KUKA KRL data list: ps_a_etb_res_c02.dat

&ACCESS RVO1
&REL 18
&COMMENT Solda Atego ETB
&PARAM DISKPATH = KRC:\R1\Program\OLP
DEFDAT  ps_a_etb_res_c02
;FOLD EXTERNAL DECLARATIONS;%{PE}%MKUKATPBASIS,%CEXT,%VCOMMON,%P
;FOLD GRIPPERTECH EXT
EXT  H50 (INT  :IN,INT  :IN,INT  :IN,GRP_TYP  :IN )
;ENDFOLD (GRIPPERTECH EXT)
;FOLD SPOTTECH EXT
EXT  USERSPOT (S_COMMAND  :IN,SPOT_TYPE  :IN )
;ENDFOLD (SPOTTECH EXT)
;FOLD BASISTECH EXT;%{PE}%MKUKATPBASIS,%CEXT,%VEXT,%P
EXT  BAS (BAS_COMMAND  :IN,REAL  :IN )
DECL INT SUCCESS
;ENDFOLD (BASISTECH EXT)
;FOLD USER EXT;%{E}%MKUKATPUSER,%CEXT,%VEXT,%P
;Make your modifications here

;ENDFOLD (USER EXT)
;ENDFOLD (EXTERNAL DECLARATIONS)


DECL FDAT Fl035={TOOL_NO 3,BASE_NO 3,IPO_FRAME #BASE,POINT2[] " "}
DECL E6POS Xl035={X 584.140991,Y 789.36499,Z 1229.97498,A 158.485001,B 12.9363003,C 166.735794,S 2,T 42}
DECL LDAT LL_OLP8={VEL 2.0,ACC 100.0,APO_DIST 0.0,APO_FAC 0.0,ORI_TYP #VAR,CIRC_TYP #BASE,JERK_FAC 50.0}
DECL FDAT Fl040={TOOL_NO 3,BASE_NO 3,IPO_FRAME #BASE,POINT2[] " "}
DECL E6POS Xl040={X 565.49762,Y 693.462708,Z 1207.63196,A 154.968201,B 9.37270164,C 157.367493,S 18,T 42,E1 0.0,E2 0.0,E3 0.0,E4 0.0,E5 0.0,E6 0.0}
DECL LDAT LL_OLP9={VEL 2.0,ACC 100.0,APO_DIST 0.0,APO_FAC 0.0,ORI_TYP #VAR,CIRC_TYP #BASE,JERK_FAC 50.0}


DECL FDAT Fl045={TOOL_NO 3,BASE_NO 3,IPO_FRAME #BASE,POINT2[] " "}
DECL E6POS Xl045={X 561.989014,Y 691.565002,Z 1096.26794,A 154.969498,B 9.37310028,C 147.3685,S 2,T 42}



DECL LDAT LL_OLP10={VEL 2.0,ACC 100.0,APO_DIST 0.0,APO_FAC 0.0,ORI_TYP #VAR,CIRC_TYP #BASE,JERK_FAC 50.0}
DECL FDAT Fl050={TOOL_NO 3,BASE_NO 3,IPO_FRAME #BASE,POINT2[] " "}
DECL E6POS Xl050={X 563.752014,Y 1566.71301,Z 1132.11096,A 154.969406,B 9.37310028,C 157.3685,S 2,T 42}


DECL LDAT LL_OLP11={VEL 2.0,ACC 100.0,APO_DIST 0.0,APO_FAC 0.0,ORI_TYP #VAR,CIRC_TYP #BASE,JERK_FAC 50.0}
DECL FDAT Fl055={TOOL_NO 3,BASE_NO 3,IPO_FRAME #BASE,POINT2[] " "}
DECL E6POS Xl055={X 878.794006,Y 1301.91504,Z 1209.96802,A -149.936798,B -80.7937012,C 61.0237007,S 2,T 34}
DECL LDAT LL_OLP12={VEL 2.0,ACC 100.0,APO_DIST 0.0,APO_FAC 0.0,ORI_TYP #VAR,CIRC_TYP #BASE,JERK_FAC 50.0}



DECL FDAT Fl060={TOOL_NO 3,BASE_NO 3,IPO_FRAME #BASE,POINT2[] " "}
DECL E6POS Xl060={X 618.291992,Y 968.916992,Z 1209.96594,A -149.936798,B -80.7937012,C 61.0236015,S 2,T 34}
DECL FDAT Fl065={TOOL_NO 3,BASE_NO 3,IPO_FRAME #BASE,POINT2[] " "}
DECL E6POS Xl065={X 584.655212,Y 961.50769,Z 1277.37,A -132.780594,B -83.9849777,C 40.2847786,S 18,T 34,E1 0.0,E2 0.0,E3 0.0,E4 0.0,E5 0.0,E6 0.0}
DECL LDAT LL_OLP14={VEL 2.0,ACC 100.0,APO_DIST 0.0,APO_FAC 0.0,ORI_TYP #VAR,CIRC_TYP #BASE,JERK_FAC 50.0}
DECL FDAT FSWP_60_7788={TOOL_NO 3,BASE_NO 3,IPO_FRAME #BASE,POINT2[] " "}
DECL E6POS XSWP_60_7788={X 594.593811,Y 987.688477,Z 1318.20203,A -158.479996,B -86.9590912,C 65.2634201,S 18,T 34,E1 0.0,E2 0.0,E3 0.0,E4 0.0,E5 0.0,E6 0.0}
DECL LDAT LL_OLP15={VEL 2.0,ACC 100.0,APO_DIST 0.0,APO_FAC 0.0,ORI_TYP #VAR,CIRC_TYP #BASE,JERK_FAC 50.0}
DECL FDAT FSWP_60_7790={TOOL_NO 3,BASE_NO 3,IPO_FRAME #BASE,POINT2[] " ",TQ_STATE FALSE}
DECL E6POS XSWP_60_7790={X 630.833008,Y 988.158813,Z 1320.07104,A 140.789505,B -87.3468933,C 128.901794,S 18,T 34,E1 0.0,E2 0.0,E3 0.0,E4 0.0,E5 0.0,E6 0.0}
DECL LDAT LL_OLP16={VEL 2.0,ACC 100.0,APO_DIST 0.0,APO_FAC 0.0,ORI_TYP #VAR,CIRC_TYP #BASE,JERK_FAC 50.0}
DECL FDAT FSWP_60_7792={TOOL_NO 3,BASE_NO 3,IPO_FRAME #BASE,POINT2[] " "}
DECL E6POS XSWP_60_7792={X 662.220581,Y 987.874329,Z 1321.43994,A 149.062607,B -87.5677567,C 121.765297,S 18,T 34,E1 0.0,E2 0.0,E3 0.0,E4 0.0,E5 0.0,E6 0.0}
DECL LDAT LL_OLP17={VEL 2.0,ACC 100.0,APO_DIST 0.0,APO_FAC 0.0,ORI_TYP #VAR,CIRC_TYP #BASE,JERK_FAC 50.0}
DECL FDAT Fl070={TOOL_NO 3,BASE_NO 3,IPO_FRAME #BASE,POINT2[] " "}
DECL E6POS Xl070={X 658.477173,Y 977.694092,Z 1301.79004,A -86.9980698,B -85.4011383,C -5.58326817,S 18,T 34,E1 0.0,E2 0.0,E3 0.0,E4 0.0,E5 0.0,E6 0.0}
DECL LDAT LL_OLP18={VEL 2.0,ACC 100.0,APO_DIST 0.0,APO_FAC 0.0,ORI_TYP #VAR,CIRC_TYP #BASE,JERK_FAC 50.0}

DECL FDAT Fl075={TOOL_NO 3,BASE_NO 3,IPO_FRAME #BASE,POINT2[] " "}



DECL E6POS Xl075={X 670.585022,Y 967.37323,Z 1219.30298,A -89.5080719,B -85.5535965,C 0.906028271,S 18,T 34,E1 0.0,E2 0.0,E3 0.0,E4 0.0,E5 0.0,E6 0.0}
DECL LDAT LL_OLP19={VEL 2.0,ACC 100.0,APO_DIST 10.0,APO_FAC 0.0,ORI_TYP #VAR,CIRC_TYP #BASE,JERK_FAC 50.0}






DECL FDAT Fl080={TOOL_NO 3,BASE_NO 3,IPO_FRAME #BASE,POINT2[] " "}
DECL E6POS Xl080={X 704.95752,Y 967.856384,Z 1264.87,A -14.49963,B -74.4627228,C -73.6447296,S 18,T 34,E1 0.0,E2 0.0,E3 0.0,E4 0.0,E5 0.0,E6 0.0}
DECL LDAT LL_OLP20={VEL 2.0,ACC 100.0,APO_DIST 10.0,APO_FAC 0.0,ORI_TYP #VAR,CIRC_TYP #BASE,JERK_FAC 50.0}
DECL FDAT Fl085={TOOL_NO 3,BASE_NO 3,IPO_FRAME #BASE,POINT2[] " "}
DECL E6POS Xl085={X 715.177124,Y 970.295776,Z 1286.88904,A -14.4969301,B -74.4632263,C -73.6462326,S 18,T 34,E1 0.0,E2 0.0,E3 0.0,E4 0.0,E5 0.0,E6 0.0}
DECL LDAT LL_OLP21={VEL 2.0,ACC 100.0,APO_DIST 0.0,APO_FAC 0.0,ORI_TYP #VAR,CIRC_TYP #BASE,JERK_FAC 50.0}
DECL FDAT FSWP_60_7796={TOOL_NO 3,BASE_NO 3,IPO_FRAME #BASE,POINT2[] " "}
DECL E6POS XSWP_60_7796={X 735.90741,Y 986.652527,Z 1321.86902,A 8.92792034,B -75.0170135,C -96.2646103,S 18,T 34,E1 0.0,E2 0.0,E3 0.0,E4 0.0,E5 0.0,E6 0.0}
DECL LDAT LL_OLP22={VEL 2.0,ACC 100.0,APO_DIST 0.0,APO_FAC 0.0,ORI_TYP #VAR,CIRC_TYP #BASE,JERK_FAC 50.0}
DECL FDAT FSWP_60_7798={TOOL_NO 3,BASE_NO 3,IPO_FRAME #BASE,POINT2[] " "}
DECL E6POS XSWP_60_7798={X 779.640076,Y 986.603088,Z 1321.69299,A 4.67745781,B -75.0973206,C -92.1623993,S 18,T 34,E1 0.0,E2 0.0,E3 0.0,E4 0.0,E5 0.0,E6 0.0}
DECL LDAT LL_OLP23={VEL 2.0,ACC 100.0,APO_DIST 0.0,APO_FAC 0.0,ORI_TYP #VAR,CIRC_TYP #BASE,JERK_FAC 50.0}
DECL FDAT FSWP_60_7800={TOOL_NO 3,BASE_NO 3,IPO_FRAME #BASE,POINT2[] " "}
DECL E6POS XSWP_60_7800={X 825.9328,Y 985.137573,Z 1320.76904,A 4.2847209,B -75.2969131,C -91.1992035,S 18,T 34,E1 0.0,E2 0.0,E3 0.0,E4 0.0,E5 0.0,E6 0.0}
DECL LDAT LL_OLP24={VEL 2.0,ACC 100.0,APO_DIST 0.0,APO_FAC 0.0,ORI_TYP #VAR,CIRC_TYP #BASE,JERK_FAC 50.0}
DECL FDAT FSWP_60_7802={TOOL_NO 3,BASE_NO 3,IPO_FRAME #BASE,POINT2[] " "}
DECL E6POS XSWP_60_7802={X 869.143188,Y 986.01178,Z 1322.323,A -7.07776499,B -75.2145462,C -79.7799606,S 18,T 34,E1 0.0,E2 0.0,E3 0.0,E4 0.0,E5 0.0,E6 0.0}
DECL LDAT LL_OLP25={VEL 2.0,ACC 100.0,APO_DIST 0.0,APO_FAC 0.0,ORI_TYP #VAR,CIRC_TYP #BASE,JERK_FAC 50.0}
DECL FDAT FSWP_60_7804={TOOL_NO 3,BASE_NO 3,IPO_FRAME #BASE,POINT2[] " "}
DECL E6POS XSWP_60_7804={X 921.059021,Y 987.353088,Z 1322.45996,A -5.14408016,B -75.1806793,C -81.9926834,S 18,T 34,E1 0.0,E2 0.0,E3 0.0,E4 0.0,E5 0.0,E6 0.0}
DECL LDAT LL_OLP26={VEL 2.0,ACC 100.0,APO_DIST 0.0,APO_FAC 0.0,ORI_TYP #VAR,CIRC_TYP #BASE,JERK_FAC 50.0}
DECL FDAT FSWP_60_7808={TOOL_NO 3,BASE_NO 3,IPO_FRAME #BASE,POINT2[] " "}
DECL E6POS XSWP_60_7808={X 1013.84802,Y 985.960999,Z 1321.65198,A -9.0603056,B -74.9901505,C -78.2635727,S 18,T 34,E1 0.0,E2 0.0,E3 0.0,E4 0.0,E5 0.0,E6 0.0}
DECL LDAT LL_OLP27={VEL 2.0,ACC 100.0,APO_DIST 0.0,APO_FAC 0.0,ORI_TYP #VAR,CIRC_TYP #BASE,JERK_FAC 50.0}
DECL FDAT FSWP_60_7810={TOOL_NO 3,BASE_NO 3,IPO_FRAME #BASE,POINT2[] " "}
DECL E6POS XSWP_60_7810={X 1060.09204,Y 986.898987,Z 1321.53003,A -9.69570732,B -74.9384232,C -77.7038574,S 18,T 34,E1 0.0,E2 0.0,E3 0.0,E4 0.0,E5 0.0,E6 0.0}
DECL LDAT LL_OLP28={VEL 2.0,ACC 100.0,APO_DIST 0.0,APO_FAC 0.0,ORI_TYP #VAR,CIRC_TYP #BASE,JERK_FAC 50.0}
DECL FDAT FSWP_60_7812={TOOL_NO 3,BASE_NO 3,IPO_FRAME #BASE,POINT2[] " "}
DECL E6POS XSWP_60_7812={X 1103.44104,Y 986.481995,Z 1321.01294,A -11.51863,B -74.7812805,C -76.1086578,S 18,T 34,E1 0.0,E2 0.0,E3 0.0,E4 0.0,E5 0.0,E6 0.0}
DECL LDAT LL_OLP29={VEL 2.0,ACC 100.0,APO_DIST 0.0,APO_FAC 0.0,ORI_TYP #VAR,CIRC_TYP #BASE,JERK_FAC 50.0}
DECL FDAT FSWP_60_7814={TOOL_NO 3,BASE_NO 3,IPO_FRAME #BASE,POINT2[] " "}
DECL E6POS XSWP_60_7814={X 1146.948,Y 986.203918,Z 1319.48206,A -9.90011024,B -74.91008,C -77.5603333,S 18,T 34,E1 0.0,E2 0.0,E3 0.0,E4 0.0,E5 0.0,E6 0.0}
DECL LDAT LL_OLP30={VEL 2.0,ACC 100.0,APO_DIST 0.0,APO_FAC 0.0,ORI_TYP #VAR,CIRC_TYP #BASE,JERK_FAC 50.0}
DECL FDAT FSWP_60_7816={TOOL_NO 3,BASE_NO 3,IPO_FRAME #BASE,POINT2[] " "}
DECL E6POS XSWP_60_7816={X 1193.84399,Y 985.979675,Z 1318.43506,A -3.22997093,B -75.0365219,C -84.5187073,S 18,T 34,E1 0.0,E2 0.0,E3 0.0,E4 0.0,E5 0.0,E6 0.0}
DECL LDAT LL_OLP31={VEL 2.0,ACC 100.0,APO_DIST 0.0,APO_FAC 0.0,ORI_TYP #VAR,CIRC_TYP #BASE,JERK_FAC 50.0}
DECL FDAT Fl090={TOOL_NO 3,BASE_NO 3,IPO_FRAME #BASE,POINT2[] " "}
DECL E6POS Xl090={X 1197.92505,Y 977.659119,Z 1291.51294,A -14.5019197,B -74.4627228,C -73.6420135,S 18,T 34,E1 0.0,E2 0.0,E3 0.0,E4 0.0,E5 0.0,E6 0.0}
DECL LDAT LL_OLP32={VEL 2.0,ACC 100.0,APO_DIST 0.0,APO_FAC 0.0,ORI_TYP #VAR,CIRC_TYP #BASE,JERK_FAC 50.0}
DECL FDAT Fl095={TOOL_NO 3,BASE_NO 3,IPO_FRAME #BASE,POINT2[] " "}
DECL E6POS Xl095={X 1176.53894,Y 994.848877,Z 1208.64905,A -44.5544205,B -83.8928528,C -43.9489098,S 18,T 34,E1 0.0,E2 0.0,E3 0.0,E4 0.0,E5 0.0,E6 0.0}
DECL LDAT LL_OLP33={VEL 2.0,ACC 100.0,APO_DIST 0.0,APO_FAC 0.0,ORI_TYP #VAR,CIRC_TYP #BASE,JERK_FAC 50.0}















DECL FDAT Fl100={TOOL_NO 3,BASE_NO 3,IPO_FRAME #BASE,POINT2[] " "}
DECL E6POS Xl100={X 795.249023,Y 1246.63,Z 1059.69897,A -149.936401,B -80.7937012,C 61.023201,S 2,T 34}
DECL LDAT LL_OLP34={VEL 2.0,ACC 100.0,APO_DIST 10.0,APO_FAC 0.0,ORI_TYP #VAR,CIRC_TYP #BASE,JERK_FAC 50.0}
DECL FDAT Fl105={TOOL_NO 3,BASE_NO 3,IPO_FRAME #BASE,POINT2[] " "}
DECL E6POS Xl105={X 1304.354,Y 1333.35901,Z 23.5259991,A 180.0,B -37.3134003,C 90.0,S 2,T 34}
DECL LDAT LL_OLP35={VEL 2.0,ACC 100.0,APO_DIST 30.0,APO_FAC 0.0,ORI_TYP #VAR,CIRC_TYP #BASE,JERK_FAC 50.0}

DECL FDAT Fl120={TOOL_NO 3,BASE_NO 3,IPO_FRAME #BASE,POINT2[] " "}

DECL E6POS Xl120={X 1303.89905,Y 1020.01202,Z 107.1138,A 179.976105,B -22.3131905,C 89.996582,S 18,T 34,E1 0.0,E2 0.0,E3 0.0,E4 0.0,E5 0.0,E6 0.0}
DECL LDAT LL_OLP38={VEL 2.0,ACC 100.0,APO_DIST 0.0,APO_FAC 0.0,ORI_TYP #VAR,CIRC_TYP #BASE,JERK_FAC 50.0}

DECL FDAT FSWP_60_7488={TOOL_NO 3,BASE_NO 3,IPO_FRAME #BASE,POINT2[] " "}

DECL E6POS XSWP_60_7488={X 1311.29602,Y 1033.21301,Z 114.044098,A 179.174393,B -22.3031502,C 90.7230225,S 18,T 34,E1 0.0,E2 0.0,E3 0.0,E4 0.0,E5 0.0,E6 0.0}
DECL LDAT LL_OLP39={VEL 2.0,ACC 100.0,APO_DIST 0.0,APO_FAC 0.0,ORI_TYP #VAR,CIRC_TYP #BASE,JERK_FAC 50.0}

DECL FDAT FSWP_60_7490={TOOL_NO 3,BASE_NO 3,IPO_FRAME #BASE,POINT2[] " "}

DECL E6POS XSWP_60_7490={X 1343.07202,Y 1031.32202,Z 114.458504,A 179.979507,B -22.3129196,C 90.9136505,S 18,T 34,E1 0.0,E2 0.0,E3 0.0,E4 0.0,E5 0.0,E6 0.0}
DECL LDAT LL_OLP40={VEL 2.0,ACC 100.0,APO_DIST 0.0,APO_FAC 0.0,ORI_TYP #VAR,CIRC_TYP #BASE,JERK_FAC 50.0}

DECL FDAT FSWP_60_7492={TOOL_NO 3,BASE_NO 3,IPO_FRAME #BASE,POINT2[] " "}

DECL E6POS XSWP_60_7492={X 1374.18799,Y 1032.23499,Z 114.821899,A -179.808701,B -22.2939205,C 89.9696426,S 18,T 34,E1 0.0,E2 0.0,E3 0.0,E4 0.0,E5 0.0,E6 0.0}
DECL LDAT LL_OLP41={VEL 2.0,ACC 100.0,APO_DIST 0.0,APO_FAC 0.0,ORI_TYP #VAR,CIRC_TYP #BASE,JERK_FAC 50.0}

DECL FDAT Fl125={TOOL_NO 3,BASE_NO 3,IPO_FRAME #BASE,POINT2[] " "}


DECL E6POS Xl125={X 1397.44604,Y 1024.76294,Z 95.6467438,A 179.9758,B -17.5534992,C 89.9962769,S 18,T 34,E1 0.0,E2 0.0,E3 0.0,E4 0.0,E5 0.0,E6 0.0}
DECL LDAT LL_OLP42={VEL 2.0,ACC 100.0,APO_DIST 0.0,APO_FAC 0.0,ORI_TYP #VAR,CIRC_TYP #BASE,JERK_FAC 50.0}
DECL FDAT Fl130={TOOL_NO 3,BASE_NO 3,IPO_FRAME #BASE,POINT2[] " "}
DECL E6POS Xl130={X 1469.67896,Y 1023.99103,Z 98.598999,A 179.975601,B -17.0133991,C 89.9968033,S 2,T 34}
DECL LDAT LL_OLP43={VEL 2.0,ACC 100.0,APO_DIST 0.0,APO_FAC 0.0,ORI_TYP #VAR,CIRC_TYP #BASE,JERK_FAC 50.0}



DECL FDAT FSWP_60_7496={TOOL_NO 3,BASE_NO 3,IPO_FRAME #BASE,POINT2[] " "}

DECL E6POS XSWP_60_7496={X 1451.85803,Y 1028.74304,Z 116.249001,A 179.984207,B -21.8110695,C 94.6477966,S 18,T 42,E1 0.0,E2 0.0,E3 0.0,E4 0.0,E5 0.0,E6 0.0}
DECL LDAT LL_OLP44={VEL 2.0,ACC 100.0,APO_DIST 0.0,APO_FAC 0.0,ORI_TYP #VAR,CIRC_TYP #BASE,JERK_FAC 50.0}

DECL FDAT FSWP_60_7498={TOOL_NO 3,BASE_NO 3,IPO_FRAME #BASE,POINT2[] " "}


DECL E6POS XSWP_60_7498={X 1491.27698,Y 1028.06201,Z 116.260399,A 179.982605,B -21.8108807,C 94.0462494,S 18,T 42,E1 0.0,E2 0.0,E3 0.0,E4 0.0,E5 0.0,E6 0.0}
DECL LDAT LL_OLP45={VEL 2.0,ACC 100.0,APO_DIST 0.0,APO_FAC 0.0,ORI_TYP #VAR,CIRC_TYP #BASE,JERK_FAC 50.0}
DECL FDAT FSWP_60_7500={TOOL_NO 3,BASE_NO 3,IPO_FRAME #BASE,POINT2[] " "}
DECL E6POS XSWP_60_7500={X 1538.92004,Y 1026.06396,Z 113.879898,A -179.763596,B -29.0331993,C 93.614418,S 18,T 34,E1 0.0,E2 0.0,E3 0.0,E4 0.0,E5 0.0,E6 0.0}
DECL LDAT LL_OLP46={VEL 2.0,ACC 100.0,APO_DIST 0.0,APO_FAC 0.0,ORI_TYP #VAR,CIRC_TYP #BASE,JERK_FAC 50.0}

DECL FDAT Fl140={TOOL_NO 3,BASE_NO 3,IPO_FRAME #BASE,POINT2[] " "}
DECL PDAT PP_OLP2={VEL 100.0,ACC 100.0,APO_DIST 0.0,APO_MODE #CDIS}
DECL E6POS Xl140={X 1610.60205,Y 1139.57495,Z 45.987999,A 179.975998,B -22.3132992,C 89.9968033,S 2,T 34}
DECL BASIS_SUGG_T LAST_BASIS={POINT1[] "PS01010001              ",POINT2[] "PS01010001              ",CP_PARAMS[] "CPDAT0                  ",PTP_PARAMS[] "PDAT0                   ",CONT[] "                        ",CP_VEL[] "2                       ",PTP_VEL[] " 100                    ",SPL_NAME[] "S0                      "}
DECL PDAT PP_OLP4={VEL 100.0,ACC 100.0,APO_DIST 30.0,APO_MODE #CDIS}
DECL E6POS Xl006={X 1083.797,Y 1451.30701,Z 836.236023,A 174.173294,B -30.1965008,C 118.184799,S 2,T 42}
DECL FDAT Fl006={TOOL_NO 3,BASE_NO 3,IPO_FRAME #BASE,POINT2[] " "}
DECL E6POS Xl011={X 563.747314,Y 1566.72302,Z 1132.10205,A 154.969299,B 9.37345028,C 157.368103,S 18,T 42,E1 0.0,E2 0.0,E3 0.0,E4 0.0,E5 0.0,E6 0.0}
DECL FDAT Fl011={TOOL_NO 3,BASE_NO 3,IPO_FRAME #BASE,POINT2[] " ",TQ_STATE FALSE}
DECL LDAT LL_OLP49={VEL 2.0,ACC 100.0,APO_DIST 0.0,APO_FAC 0.0,ORI_TYP #VAR,CIRC_TYP #BASE,JERK_FAC 50.0}
DECL E6POS Xl016={X 561.989014,Y 691.565002,Z 1096.26794,A 154.969498,B 9.37310028,C 147.3685,S 2,T 42}
DECL FDAT Fl016={TOOL_NO 3,BASE_NO 3,IPO_FRAME #BASE,POINT2[] " "}
DECL PDAT PP_OLP5={VEL 100.0,ACC 100.0,APO_DIST 0.0}
DECL E6POS Xl021={X 563.750977,Y 693.715027,Z 1132.11096,A 154.969406,B 9.37310028,C 157.3685,S 2,T 42}
DECL FDAT Fl021={TOOL_NO 3,BASE_NO 3,IPO_FRAME #BASE,POINT2[] " "}
DECL LDAT LL_OLP50={VEL 2.0,ACC 100.0,APO_DIST 30.0,APO_FAC 0.0,ORI_TYP #VAR,CIRC_TYP #BASE,JERK_FAC 50.0}
DECL E6POS Xl026={X 584.140991,Y 789.36499,Z 1229.97498,A 158.485001,B 12.9363003,C 166.735794,S 2,T 42}
DECL FDAT Fl026={TOOL_NO 3,BASE_NO 3,IPO_FRAME #BASE,POINT2[] " "}












DECL LDAT LL_OLP51={VEL 2.0,ACC 100.0,APO_DIST 0.0,APO_FAC 0.0,ORI_TYP #VAR,CIRC_TYP #BASE,JERK_FAC 50.0}
DECL E6POS Xl031={X 349.9328,Y 278.265503,Z 1120.06702,A 150.3909,B 43.1627502,C 155.956406,S 18,T 42,E1 0.0,E2 0.0,E3 0.0,E4 0.0,E5 0.0,E6 0.0}
DECL FDAT Fl031={TOOL_NO 3,BASE_NO 3,IPO_FRAME #BASE,POINT2[] " "}
DECL PDAT PP_OLP6={VEL 100.0,ACC 100.0,APO_DIST 0.0}
DECL E6POS Xl036={X 305.381195,Y 288.633514,Z 1051.12598,A 147.643494,B 47.8914604,C 153.831299,S 18,T 42,E1 0.0,E2 0.0,E3 0.0,E4 0.0,E5 0.0,E6 0.0}
DECL FDAT Fl036={TOOL_NO 3,BASE_NO 3,IPO_FRAME #BASE,POINT2[] " "}
DECL PDAT PP_OLP7={VEL 100.0,ACC 100.0,APO_DIST 10.0,APO_MODE #CDIS}
DECL E6POS Xl041={X 103.434502,Y 364.44751,Z 683.522705,A 164.801605,B 79.9912796,C 167.123993,S 18,T 42,E1 0.0,E2 0.0,E3 0.0,E4 0.0,E5 0.0,E6 0.0}
DECL FDAT Fl041={TOOL_NO 3,BASE_NO 3,IPO_FRAME #BASE,POINT2[] " "}
DECL LDAT LL_OLP52={VEL 2.0,ACC 100.0,APO_DIST 0.0,APO_FAC 0.0,ORI_TYP #VAR,CIRC_TYP #BASE,JERK_FAC 50.0}
DECL E6POS Xl046={X 91.8286896,Y 379.290894,Z 653.815796,A 159.358994,B 82.8835907,C 161.735306,S 18,T 42,E1 0.0,E2 0.0,E3 0.0,E4 0.0,E5 0.0,E6 0.0}
DECL FDAT Fl046={TOOL_NO 3,BASE_NO 3,IPO_FRAME #BASE,POINT2[] " "}
DECL LDAT LL_OLP53={VEL 2.0,ACC 100.0,APO_DIST 0.0,APO_FAC 0.0,ORI_TYP #VAR,CIRC_TYP #BASE,JERK_FAC 50.0}
DECL E6POS XSWP_60_7880={X 93.7982178,Y 380.760986,Z 613.06543,A 159.360794,B 82.8838272,C 161.736404,S 18,T 42,E1 0.0,E2 0.0,E3 0.0,E4 0.0,E5 0.0,E6 0.0}
DECL FDAT FSWP_60_7880={TOOL_NO 3,BASE_NO 3,IPO_FRAME #BASE,POINT2[] " "}
DECL LDAT LL_OLP54={VEL 2.0,ACC 100.0,APO_DIST 0.0,APO_FAC 0.0,ORI_TYP #VAR,CIRC_TYP #BASE,JERK_FAC 50.0}
DECL E6POS XSWP_60_7882={X 95.1983414,Y 412.033203,Z 612.224121,A 159.370499,B 82.8822937,C 161.745895,S 18,T 42,E1 0.0,E2 0.0,E3 0.0,E4 0.0,E5 0.0,E6 0.0}
DECL FDAT FSWP_60_7882={TOOL_NO 3,BASE_NO 3,IPO_FRAME #BASE,POINT2[] " "}
DECL LDAT LL_OLP55={VEL 2.0,ACC 100.0,APO_DIST 0.0,APO_FAC 0.0,ORI_TYP #VAR,CIRC_TYP #BASE,JERK_FAC 50.0}
DECL E6POS XSWP_60_7886={X 98.8377228,Y 478.136993,Z 615.090515,A 158.5354,B 82.6687012,C 159.334305,S 18,T 42,E1 0.0,E2 0.0,E3 0.0,E4 0.0,E5 0.0,E6 0.0}
DECL FDAT FSWP_60_7886={TOOL_NO 3,BASE_NO 3,IPO_FRAME #BASE,POINT2[] " "}
DECL LDAT LL_OLP56={VEL 2.0,ACC 100.0,APO_DIST 0.0,APO_FAC 0.0,ORI_TYP #VAR,CIRC_TYP #BASE,JERK_FAC 50.0}
DECL E6POS XSWP_60_7888={X 100.442497,Y 513.4646,Z 616.12793,A 159.082596,B 82.9018936,C 159.794601,S 18,T 42,E1 0.0,E2 0.0,E3 0.0,E4 0.0,E5 0.0,E6 0.0}
DECL FDAT FSWP_60_7888={TOOL_NO 3,BASE_NO 3,IPO_FRAME #BASE,POINT2[] " "}
DECL LDAT LL_OLP57={VEL 2.0,ACC 100.0,APO_DIST 0.0,APO_FAC 0.0,ORI_TYP #VAR,CIRC_TYP #BASE,JERK_FAC 50.0}
DECL E6POS XSWP_60_7990={X 102.522003,Y 545.988403,Z 614.039917,A 160.234299,B 82.879837,C 161.132095,S 18,T 42,E1 0.0,E2 0.0,E3 0.0,E4 0.0,E5 0.0,E6 0.0}
DECL FDAT FSWP_60_7990={TOOL_NO 3,BASE_NO 3,IPO_FRAME #BASE,POINT2[] " "}
DECL LDAT LL_OLP58={VEL 2.0,ACC 100.0,APO_DIST 0.0,APO_FAC 0.0,ORI_TYP #VAR,CIRC_TYP #BASE,JERK_FAC 50.0}
DECL E6POS XSWP_60_7892={X 103.919098,Y 574.488892,Z 615.100891,A 159.7061,B 82.8799286,C 161.684998,S 18,T 42,E1 0.0,E2 0.0,E3 0.0,E4 0.0,E5 0.0,E6 0.0}
DECL FDAT FSWP_60_7892={TOOL_NO 3,BASE_NO 3,IPO_FRAME #BASE,POINT2[] " "}
DECL LDAT LL_OLP59={VEL 2.0,ACC 100.0,APO_DIST 0.0,APO_FAC 0.0,ORI_TYP #VAR,CIRC_TYP #BASE,JERK_FAC 50.0}
DECL E6POS XSWP_60_7896={X 108.416,Y 646.456177,Z 614.435181,A 159.410507,B 82.8830185,C 161.785904,S 18,T 42,E1 0.0,E2 0.0,E3 0.0,E4 0.0,E5 0.0,E6 0.0}
DECL FDAT FSWP_60_7896={TOOL_NO 3,BASE_NO 3,IPO_FRAME #BASE,POINT2[] " "}
DECL LDAT LL_OLP60={VEL 2.0,ACC 100.0,APO_DIST 0.0,APO_FAC 0.0,ORI_TYP #VAR,CIRC_TYP #BASE,JERK_FAC 50.0}
DECL E6POS XSWP_60_7898={X 111.716202,Y 682.766418,Z 615.322815,A 159.398407,B 82.8831482,C 161.775604,S 18,T 42,E1 0.0,E2 0.0,E3 0.0,E4 0.0,E5 0.0,E6 0.0}
DECL FDAT FSWP_60_7898={TOOL_NO 3,BASE_NO 3,IPO_FRAME #BASE,POINT2[] " "}
DECL LDAT LL_OLP61={VEL 2.0,ACC 100.0,APO_DIST 0.0,APO_FAC 0.0,ORI_TYP #VAR,CIRC_TYP #BASE,JERK_FAC 50.0}
DECL E6POS XSWP_60_7900={X 114.766197,Y 718.722412,Z 616.54657,A 159.434402,B 82.8802872,C 161.813995,S 18,T 42,E1 0.0,E2 0.0,E3 0.0,E4 0.0,E5 0.0,E6 0.0}
DECL FDAT FSWP_60_7900={TOOL_NO 3,BASE_NO 3,IPO_FRAME #BASE,POINT2[] " "}
DECL LDAT LL_OLP62={VEL 2.0,ACC 100.0,APO_DIST 0.0,APO_FAC 0.0,ORI_TYP #VAR,CIRC_TYP #BASE,JERK_FAC 50.0}
DECL E6POS XSWP_60_7902={X 119.6847,Y 754.768677,Z 617.763794,A 159.414795,B 82.8860092,C 161.790604,S 18,T 42,E1 0.0,E2 0.0,E3 0.0,E4 0.0,E5 0.0,E6 0.0}
DECL FDAT FSWP_60_7902={TOOL_NO 3,BASE_NO 3,IPO_FRAME #BASE,POINT2[] " "}
DECL LDAT LL_OLP63={VEL 2.0,ACC 100.0,APO_DIST 0.0,APO_FAC 0.0,ORI_TYP #VAR,CIRC_TYP #BASE,JERK_FAC 50.0}
DECL E6POS XSWP_60_7904={X 124.1399,Y 792.107971,Z 618.820129,A 159.417999,B 82.8863525,C 161.793106,S 18,T 42,E1 0.0,E2 0.0,E3 0.0,E4 0.0,E5 0.0,E6 0.0}
DECL FDAT FSWP_60_7904={TOOL_NO 3,BASE_NO 3,IPO_FRAME #BASE,POINT2[] " "}
DECL LDAT LL_OLP64={VEL 2.0,ACC 100.0,APO_DIST 0.0,APO_FAC 0.0,ORI_TYP #VAR,CIRC_TYP #BASE,JERK_FAC 50.0}
DECL E6POS XSWP_60_7906={X 132.870697,Y 841.648804,Z 621.361816,A 159.395203,B 82.8851624,C 161.773804,S 18,T 42,E1 0.0,E2 0.0,E3 0.0,E4 0.0,E5 0.0,E6 0.0}
DECL FDAT FSWP_60_7906={TOOL_NO 3,BASE_NO 3,IPO_FRAME #BASE,POINT2[] " "}
DECL LDAT LL_OLP65={VEL 2.0,ACC 100.0,APO_DIST 0.0,APO_FAC 0.0,ORI_TYP #VAR,CIRC_TYP #BASE,JERK_FAC 50.0}
DECL E6POS XSWP_60_7908={X 139.911102,Y 879.169617,Z 618.96582,A 159.404099,B 82.897049,C 167.300797,S 18,T 42,E1 0.0,E2 0.0,E3 0.0,E4 0.0,E5 0.0,E6 0.0}
DECL FDAT FSWP_60_7908={TOOL_NO 3,BASE_NO 3,IPO_FRAME #BASE,POINT2[] " "}
DECL E6POS Xl051={X 137.945007,Y 854.049988,Z 676.479004,A 164.794098,B 79.9898987,C 167.113907,S 2,T 42}
DECL FDAT Fl051={TOOL_NO 3,BASE_NO 3,IPO_FRAME #BASE,POINT2[] " "}
DECL SPOT_TYPE SNORMAL={GUN 1,PAIR #FIRST,RETR #OPN,CLO_TM 0,PGNO1 1,PRESS1 0.0,PGNO2 0,PRESS2 0.0}
DECL E6POS XP3={X 567.326416,Y 409.623993,Z 1234.31702,A 158.465195,B 12.93505,C 166.748199,S 18,T 42,E1 0.0,E2 0.0,E3 0.0,E4 0.0,E5 0.0,E6 0.0}
DECL FDAT FP3={TOOL_NO 3,BASE_NO 3,IPO_FRAME #BASE,POINT2[] " ",TQ_STATE FALSE}
DECL LDAT LCPDAT2={VEL 2.0,ACC 100.0,APO_DIST 10.0,APO_FAC 50.0,AXIS_VEL 100.0,AXIS_ACC 100.0,ORI_TYP #VAR,CIRC_TYP #BASE,JERK_FAC 50.0,GEAR_JERK 50.0,EXAX_IGN 0}
DECL E6POS XP6={X 558.674316,Y 257.743713,Z 1366.94299,A 155.132797,B 22.3248005,C 163.028503,S 18,T 42,E1 0.0,E2 0.0,E3 0.0,E4 0.0,E5 0.0,E6 0.0}
DECL FDAT FP6={TOOL_NO 3,BASE_NO 3,IPO_FRAME #BASE,POINT2[] " ",TQ_STATE FALSE}
DECL LDAT LCPDAT5={VEL 2.0,ACC 100.0,APO_DIST 100.0,APO_FAC 50.0,AXIS_VEL 100.0,AXIS_ACC 100.0,ORI_TYP #VAR,CIRC_TYP #BASE,JERK_FAC 50.0,GEAR_JERK 50.0,EXAX_IGN 0}
DECL E6POS XP7={X 622.916321,Y 355.254211,Z 1422.57605,A 157.948105,B 12.9317598,C 166.758606,S 18,T 42,E1 0.0,E2 0.0,E3 0.0,E4 0.0,E5 0.0,E6 0.0}
DECL FDAT FP7={TOOL_NO 3,BASE_NO 3,IPO_FRAME #BASE,POINT2[] " ",TQ_STATE FALSE}
DECL LDAT LCPDAT6={VEL 2.0,ACC 100.0,APO_DIST 100.0,APO_FAC 50.0,AXIS_VEL 100.0,AXIS_ACC 100.0,ORI_TYP #VAR,CIRC_TYP #BASE,JERK_FAC 50.0,GEAR_JERK 50.0,EXAX_IGN 0}
DECL E6POS XP8={X 407.655396,Y 277.337799,Z 1190.83606,A 150.367401,B 35.5736084,C 156.603897,S 18,T 42,E1 0.0,E2 0.0,E3 0.0,E4 0.0,E5 0.0,E6 0.0}
DECL FDAT FP8={TOOL_NO 3,BASE_NO 3,IPO_FRAME #BASE,POINT2[] " ",TQ_STATE FALSE}
DECL LDAT LCPDAT7={VEL 2.0,ACC 100.0,APO_DIST 100.0,APO_FAC 50.0,AXIS_VEL 100.0,AXIS_ACC 100.0,ORI_TYP #VAR,CIRC_TYP #BASE,JERK_FAC 50.0,GEAR_JERK 50.0,EXAX_IGN 0}


DECL E6POS XP11={X 1560.58704,Y 1009.72302,Z 65.5483475,A 179.964401,B -43.8393517,C 90.9567795,S 18,T 34,E1 0.0,E2 0.0,E3 0.0,E4 0.0,E5 0.0,E6 0.0}
DECL FDAT FP11={TOOL_NO 3,BASE_NO 3,IPO_FRAME #BASE,POINT2[] " ",TQ_STATE FALSE}

DECL LDAT LCPDAT10={VEL 2.0,ACC 100.0,APO_DIST 100.0,APO_FAC 50.0,AXIS_VEL 100.0,AXIS_ACC 100.0,ORI_TYP #VAR,CIRC_TYP #BASE,JERK_FAC 50.0,GEAR_JERK 50.0,EXAX_IGN 0}
DECL SPOT_SUGG_T LAST_SPOT={GUN[] "1                       ",RETR_CMD[] "#OPN                    ",CHOISE[] "#FIRST                  ",CLO_TM[] "0                       ",PGNO1[] "1                       ",PRESS1[] "0                       ",PGNO2[] "1                       ",PRESS2[] "0                       ",SPOT_PARAMS[] "NORMAL                  "}
DECL E6POS XP14={X 1610.68799,Y 1340.54297,Z 45.7100296,A 179.967102,B -22.3057804,C 90.001152,S 18,T 34,E1 0.0,E2 0.0,E3 0.0,E4 0.0,E5 0.0,E6 0.0}
DECL FDAT FP14={TOOL_NO 3,BASE_NO 3,IPO_FRAME #BASE,POINT2[] " ",TQ_STATE FALSE}
DECL PDAT PPDAT5={VEL 100.0,ACC 95.0,APO_DIST 100.0,APO_MODE #CDIS,GEAR_JERK 50.0}
DECL E6POS XP16={X 1711.52502,Y 2023.51099,Z 556.947876,A -175.166397,B -41.1158485,C 86.8608398,S 18,T 34,E1 0.0,E2 0.0,E3 0.0,E4 0.0,E5 0.0,E6 0.0}
DECL FDAT FP16={TOOL_NO 3,BASE_NO 3,IPO_FRAME #BASE,POINT2[] " ",TQ_STATE FALSE}
DECL PDAT PPDAT7={VEL 100.0,ACC 100.0,APO_DIST 100.0,APO_MODE #CDIS,GEAR_JERK 50.0}
DECL E6POS XP17={X 1711.651,Y 2023.50098,Z 556.917297,A -175.160202,B -41.1122093,C 86.8591003,S 18,T 42,E1 0.0,E2 0.0,E3 0.0,E4 0.0,E5 0.0,E6 0.0}


DECL FDAT FP17={TOOL_NO 3,BASE_NO 3,IPO_FRAME #BASE,POINT2[] " ",TQ_STATE FALSE}
DECL PDAT PPDAT8={VEL 100.0,ACC 100.0,APO_DIST 100.0,APO_MODE #CDIS,GEAR_JERK 50.0}
DECL LDAT LCPDAT11={VEL 2.0,ACC 100.0,APO_DIST 10.0,APO_FAC 50.0,AXIS_VEL 100.0,AXIS_ACC 100.0,ORI_TYP #VAR,CIRC_TYP #BASE,JERK_FAC 50.0,GEAR_JERK 50.0,EXAX_IGN 0}
DECL E6POS XP18={X 60.9463196,Y 487.706207,Z 619.175598,A 160.159195,B 82.8793716,C 161.610504,S 18,T 42,E1 0.0,E2 0.0,E3 0.0,E4 0.0,E5 0.0,E6 0.0}
DECL FDAT FP18={TOOL_NO 3,BASE_NO 3,IPO_FRAME #BASE,POINT2[] " ",TQ_STATE FALSE}
DECL LDAT LCPDAT12={VEL 2.0,ACC 100.0,APO_DIST 10.0,APO_FAC 50.0,AXIS_VEL 100.0,AXIS_ACC 100.0,ORI_TYP #VAR,CIRC_TYP #BASE,JERK_FAC 50.0,GEAR_JERK 50.0,EXAX_IGN 0}

DECL E6POS XP19={X 128.315308,Y 824.686523,Z 636.831726,A 156.575699,B 83.7855835,C 158.972504,S 18,T 42,E1 0.0,E2 0.0,E3 0.0,E4 0.0,E5 0.0,E6 0.0}

DECL FDAT FP19={TOOL_NO 3,BASE_NO 3,IPO_FRAME #BASE,POINT2[] " ",TQ_STATE FALSE}

DECL LDAT LL_OLP68={VEL 2.0,ACC 100.0,APO_DIST 10.0,APO_FAC 0.0,ORI_TYP #VAR,CIRC_TYP #BASE,JERK_FAC 50.0}
DECL E6POS Xl037={X 416.389008,Y 806.565979,Z 1106.76904,A 158.978607,B 33.3137093,C 165.382401,S 18,T 42,E1 0.0,E2 0.0,E3 0.0,E4 0.0,E5 0.0,E6 0.0}
DECL FDAT Fl037={TOOL_NO 3,BASE_NO 3,IPO_FRAME #BASE,POINT2[] " "}


DECL LDAT LL_OLP69={VEL 2.0,ACC 100.0,APO_DIST 0.0,APO_FAC 0.0,ORI_TYP #VAR,CIRC_TYP #BASE,JERK_FAC 50.0}
DECL E6POS XSWP_60_7346={X 145.023697,Y 915.326477,Z 621.096924,A 92.0248337,B 54.5312805,C 101.881203,S 18,T 42,E1 0.0,E2 0.0,E3 0.0,E4 0.0,E5 0.0,E6 0.0}
DECL FDAT FSWP_60_7346={TOOL_NO 3,BASE_NO 3,IPO_FRAME #BASE,POINT2[] " ",TQ_STATE FALSE}
DECL LDAT LCPDAT15={VEL 2.0,ACC 100.0,APO_DIST 5.0,APO_FAC 50.0,AXIS_VEL 100.0,AXIS_ACC 100.0,ORI_TYP #VAR,CIRC_TYP #BASE,JERK_FAC 50.0,GEAR_JERK 50.0,EXAX_IGN 0}
DECL PDAT PPDAT10={VEL 100.0,ACC 100.0,APO_DIST 30.0,APO_MODE #CDIS,GEAR_JERK 50.0}
DECL LDAT LCPDAT16={VEL 2.0,ACC 100.0,APO_DIST 30.0,APO_FAC 50.0,AXIS_VEL 100.0,AXIS_ACC 100.0,ORI_TYP #VAR,CIRC_TYP #BASE,JERK_FAC 50.0,GEAR_JERK 50.0,EXAX_IGN 0}
DECL LDAT LCPDAT0={VEL 2.0,ACC 100.0,APO_DIST 30.0,APO_FAC 50.0,AXIS_VEL 100.0,AXIS_ACC 100.0,ORI_TYP #VAR,CIRC_TYP #BASE,JERK_FAC 50.0,GEAR_JERK 50.0,EXAX_IGN 0}
DECL E6POS Xl066={X 1312.10205,Y 1148.0,Z 79.7080002,A 180.0,B -13.3133001,C 90.0,S 2,T 42}
DECL FDAT Fl066={TOOL_NO 3,BASE_NO 3,IPO_FRAME #BASE,POINT2[] " "}
DECL LDAT LCPDAT17={VEL 2.0,ACC 100.0,APO_DIST 5.0,APO_FAC 50.0,AXIS_VEL 100.0,AXIS_ACC 100.0,ORI_TYP #VAR,CIRC_TYP #BASE,JERK_FAC 50.0,GEAR_JERK 50.0,EXAX_IGN 0}
DECL E6POS XP0={X 1230.61096,Y 1015.41901,Z 62.1031799,A -179.999207,B -13.3151903,C 90.0011368,S 18,T 42,E1 0.0,E2 0.0,E3 0.0,E4 0.0,E5 0.0,E6 0.0}
DECL FDAT FP0={TOOL_NO 3,BASE_NO 3,IPO_FRAME #BASE,POINT2[] " ",TQ_STATE FALSE}
DECL LDAT LL_OLP70={VEL 2.0,ACC 100.0,APO_DIST 5.0,APO_FAC 0.0,ORI_TYP #VAR,CIRC_TYP #BASE,JERK_FAC 50.0}
DECL E6POS Xl071={X 1116.63403,Y 1017.16602,Z 51.4317093,A 179.996597,B -13.3109398,C 90.0032806,S 18,T 42,E1 0.0,E2 0.0,E3 0.0,E4 0.0,E5 0.0,E6 0.0}
DECL FDAT Fl071={TOOL_NO 3,BASE_NO 3,IPO_FRAME #BASE,POINT2[] " ",TQ_STATE FALSE}
DECL LDAT LCPDAT18={VEL 2.0,ACC 100.0,APO_DIST 5.0,APO_FAC 50.0,AXIS_VEL 100.0,AXIS_ACC 100.0,ORI_TYP #VAR,CIRC_TYP #BASE,JERK_FAC 50.0,GEAR_JERK 50.0,EXAX_IGN 0}
DECL E6POS XP21={X 1108.78296,Y 1017.35999,Z 73.2284927,A 179.996597,B -13.3102198,C 90.0024872,S 18,T 42,E1 0.0,E2 0.0,E3 0.0,E4 0.0,E5 0.0,E6 0.0}
DECL FDAT FP21={TOOL_NO 3,BASE_NO 3,IPO_FRAME #BASE,POINT2[] " ",TQ_STATE FALSE}
DECL LDAT LCPDAT19={VEL 2.0,ACC 100.0,APO_DIST 100.0,APO_FAC 50.0,AXIS_VEL 100.0,AXIS_ACC 100.0,ORI_TYP #VAR,CIRC_TYP #BASE,JERK_FAC 50.0,GEAR_JERK 50.0,EXAX_IGN 0}
DECL E6POS XSWP_61_7028={X 1103.71106,Y 1027.16394,Z 73.6532211,A 179.998795,B -13.3108597,C 90.0045013,S 18,T 42,E1 0.0,E2 0.0,E3 0.0,E4 0.0,E5 0.0,E6 0.0}
DECL FDAT FSWP_61_7028={TOOL_NO 3,BASE_NO 3,IPO_FRAME #BASE,POINT2[] " ",TQ_STATE FALSE}
DECL LDAT LCPDAT20={VEL 2.0,ACC 100.0,APO_DIST 100.0,APO_FAC 50.0,AXIS_VEL 100.0,AXIS_ACC 100.0,ORI_TYP #VAR,CIRC_TYP #BASE,JERK_FAC 50.0,GEAR_JERK 50.0,EXAX_IGN 0}
DECL E6POS XSWP_61_7030={X 1150.83301,Y 1025.60095,Z 92.6395035,A -179.999695,B -13.3080397,C 90.0064468,S 18,T 42,E1 0.0,E2 0.0,E3 0.0,E4 0.0,E5 0.0,E6 0.0}
DECL FDAT FSWP_61_7030={TOOL_NO 3,BASE_NO 3,IPO_FRAME #BASE,POINT2[] " ",TQ_STATE FALSE}
DECL LDAT LCPDAT21={VEL 2.0,ACC 100.0,APO_DIST 100.0,APO_FAC 50.0,AXIS_VEL 100.0,AXIS_ACC 100.0,ORI_TYP #VAR,CIRC_TYP #BASE,JERK_FAC 50.0,GEAR_JERK 50.0,EXAX_IGN 0}
DECL E6POS XSWP_61_7032={X 1207.69495,Y 1024.18103,Z 101.351501,A -179.906403,B -19.7679901,C 90.0272598,S 18,T 34,E1 0.0,E2 0.0,E3 0.0,E4 0.0,E5 0.0,E6 0.0}
DECL FDAT FSWP_61_7032={TOOL_NO 3,BASE_NO 3,IPO_FRAME #BASE,POINT2[] " ",TQ_STATE FALSE}
DECL LDAT LCPDAT22={VEL 2.0,ACC 100.0,APO_DIST 10.0,APO_FAC 50.0,AXIS_VEL 100.0,AXIS_ACC 100.0,ORI_TYP #VAR,CIRC_TYP #BASE,JERK_FAC 50.0,GEAR_JERK 50.0,EXAX_IGN 0}
DECL E6POS XP22={X 1206.38403,Y 1006.83502,Z 67.4408493,A -179.908997,B -19.7681408,C 90.0280304,S 18,T 34,E1 0.0,E2 0.0,E3 0.0,E4 0.0,E5 0.0,E6 0.0}
DECL FDAT FP22={TOOL_NO 3,BASE_NO 3,IPO_FRAME #BASE,POINT2[] " ",TQ_STATE FALSE}
DECL LDAT LCPDAT23={VEL 2.0,ACC 100.0,APO_DIST 10.0,APO_FAC 50.0,AXIS_VEL 100.0,AXIS_ACC 100.0,ORI_TYP #VAR,CIRC_TYP #BASE,JERK_FAC 50.0,GEAR_JERK 50.0,EXAX_IGN 0}
DECL E6POS XP23={X 1318.18396,Y 1023.573,Z 67.8225021,A 179.9785,B -22.2590103,C 89.997673,S 18,T 34,E1 0.0,E2 0.0,E3 0.0,E4 0.0,E5 0.0,E6 0.0}
DECL FDAT FP23={TOOL_NO 3,BASE_NO 3,IPO_FRAME #BASE,POINT2[] " ",TQ_STATE FALSE}
DECL E6POS XSWP_60_7890={X 102.528702,Y 545.992371,Z 614.040771,A 160.234497,B 82.8797607,C 161.132202,S 18,T 42,E1 0.0,E2 0.0,E3 0.0,E4 0.0,E5 0.0,E6 0.0}
DECL FDAT FSWP_60_7890={TOOL_NO 3,BASE_NO 3,IPO_FRAME #BASE,POINT2[] " ",TQ_STATE FALSE}
ENDDAT
